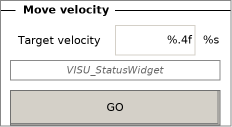
VISUALIZATION VISU_BaseAxis_MoveVelocity  // 232x127
VAR_IN_OUT
	axis : BaseAxis;
    axisWidget : BaseAxisWidget;
    positionSymbol : STRING;
    velocitySymbol : STRING;
END_VAR
    Label (15,26 100x29), "Target velocity"
    Button (10,90 210x35), "GO", input disabled if: axis.processes.moveVelocity.statuses.enabledStatus.disabled
        OnMouseClick: execute { axis.processes.moveVelocity.do_request := TRUE; }
    Line (0,10) (15,10)
    Label (20,0 150x20), "Move velocity"
    Line (115,10) (230,10)
    Textfield (115,25 80x30), "%.4f", text variable: axis.processes.moveVelocity.set.value, input disabled if: axis.processes.moveVelocity.statuses.enabledStatus.disabled
        OnMouseClick: write the text variable via VisuDialogs.Numpad
    Frame (10,60 210x20)
        shows VISU_StatusWidget(widget := axisWidget.moveVelocityProcess.actualStatus)
    Rectangle (200,25 30x30), "%s", text variable: velocitySymbol
END_VISUALIZATION

(* stored: Version 1.1.0.1, ProductVersion 3.1.4019.2
   Visu VISU_BaseAxis_MoveVelocity: Id {aebb96ca-b97f-4f5d-beb9-379362f39f9c} *)
